// TIA Portal V20 export
// export: Created 2025-12-01T14:57:42.979412Z, ExportSetting None, DisplayName Totally Integrated Automation Portal, DisplayVersion V20 Update 3, DisplayName TIA Portal Openness, DisplayVersion V20 Update 3, DisplayName TIA Portal Version Control Interface, DisplayVersion V20 Update 3, DisplayName STEP 7 Professional, DisplayVersion V20 Update 3, DisplayName STEP 7 Safety, DisplayVersion V20 Update 2, DisplayName WinCC Basic/Comfort/Advanced, DisplayVersion V20 Update 3, DisplayName WinCC Professional, DisplayVersion V20 Update 3, DisplayName WinCC Unified, DisplayVersion V20 Update 3
FUNCTION "FC954_Recoger_Diag_Gateway" : Void   // FC954, LAD
{ S7_Optimized_Access := 'TRUE' }
// stored: AutoNumber false, SetENOAutomatically false
   VAR_TEMP
      i : Int;
      indice : Int;
      datos_gateway : Struct
         Diagnosticar : Bool;   // activar el diagnosticar solo si existe
         Dos_lineas : Bool;
         hwld : HW_IO;
         Dir_ini_diag : Int;
         Dir_ini_Asi5_L1 : Int;
         Dir_ini_ASi5_L2 : Int;
      END_STRUCT;
   END_VAR
BEGIN

REGION Network 1 (SCL)
   // recoger los datos de diagnostico de todos los gateways
   // 
   FOR #indice := 1 TO 8 BY 1 DO
       IF "DB1904_Datos_Config_Gateways".Gateway[#indice].Diagnosticar = true THEN
           #datos_gateway := "DB1904_Datos_Config_Gateways".Gateway[#indice];
           REGION diagnostico_L1
               // diagnostico ASi3- Canal 1
               "DB1903_ASI_DIAG".ASI3_GW_C1[#indice]."Flags Fault Det" := PEEK_WORD(area := 16#1, dbNumber := 0, byteOffset := #datos_gateway.Dir_ini_diag);
               "DB1903_ASI_DIAG".ASI3_GW_C1[#indice].ConfigErrorsW0 := PEEK_WORD(area := 16#1, dbNumber := 0, byteOffset := (#datos_gateway.Dir_ini_diag + 2));
               "DB1903_ASI_DIAG".ASI3_GW_C1[#indice].ConfigErrorsW2 := PEEK_WORD(area := 16#1, dbNumber := 0, byteOffset := (#datos_gateway.Dir_ini_diag + 4));
               "DB1903_ASI_DIAG".ASI3_GW_C1[#indice].ConfigErrorsW4 := PEEK_WORD(area := 16#1, dbNumber := 0, byteOffset := (#datos_gateway.Dir_ini_diag + 6));
               "DB1903_ASI_DIAG".ASI3_GW_C1[#indice].ConfigErrorsW6 := PEEK_WORD(area := 16#1, dbNumber := 0, byteOffset := (#datos_gateway.Dir_ini_diag + 8));
               "DB1903_ASI_DIAG".ASI3_GW_C1[#indice].PeripheryFaultsW0 := PEEK_WORD(area := 16#1, dbNumber := 0, byteOffset := (#datos_gateway.Dir_ini_diag + 10));
               "DB1903_ASI_DIAG".ASI3_GW_C1[#indice].PeripheryFaultsW2 := PEEK_WORD(area := 16#1, dbNumber := 0, byteOffset := (#datos_gateway.Dir_ini_diag + 12));
               "DB1903_ASI_DIAG".ASI3_GW_C1[#indice].PeripheryFaultsW4 := PEEK_WORD(area := 16#1, dbNumber := 0, byteOffset := (#datos_gateway.Dir_ini_diag + 14));
               "DB1903_ASI_DIAG".ASI3_GW_C1[#indice].PeripheryFaultsW6 := PEEK_WORD(area := 16#1, dbNumber := 0, byteOffset := (#datos_gateway.Dir_ini_diag + 16));

               // diagnostico ASi5- Canal 1
               "DB1903_ASI_DIAG".ASI5_GW_C1[#indice].ConfigErrorsW0 := PEEK_WORD(area := 16#1, dbNumber := 0, byteOffset := #datos_gateway.Dir_ini_diag + 18);
               "DB1903_ASI_DIAG".ASI5_GW_C1[#indice].ConfigErrorsW2 := PEEK_WORD(area := 16#1, dbNumber := 0, byteOffset := #datos_gateway.Dir_ini_diag + 20);
               "DB1903_ASI_DIAG".ASI5_GW_C1[#indice].ConfigErrorsW4 := PEEK_WORD(area := 16#1, dbNumber := 0, byteOffset := #datos_gateway.Dir_ini_diag + 22);
               "DB1903_ASI_DIAG".ASI5_GW_C1[#indice].ConfigErrorsW6 := PEEK_WORD(area := 16#1, dbNumber := 0, byteOffset := #datos_gateway.Dir_ini_diag + 24);
               "DB1903_ASI_DIAG".ASI5_GW_C1[#indice].ConfigErrorsW8 := PEEK_WORD(area := 16#1, dbNumber := 0, byteOffset := #datos_gateway.Dir_ini_diag + 26);
               "DB1903_ASI_DIAG".ASI5_GW_C1[#indice].ConfigErrorsW10 := PEEK_WORD(area := 16#1, dbNumber := 0, byteOffset := #datos_gateway.Dir_ini_diag + 28);
               "DB1903_ASI_DIAG".ASI5_GW_C1[#indice].PeripheryFaultsW0 := PEEK_WORD(area := 16#1, dbNumber := 0, byteOffset := #datos_gateway.Dir_ini_diag + 30);
               "DB1903_ASI_DIAG".ASI5_GW_C1[#indice].PeripheryFaultsW2 := PEEK_WORD(area := 16#1, dbNumber := 0, byteOffset := #datos_gateway.Dir_ini_diag + 32);
               "DB1903_ASI_DIAG".ASI5_GW_C1[#indice].PeripheryFaultsW4 := PEEK_WORD(area := 16#1, dbNumber := 0, byteOffset := #datos_gateway.Dir_ini_diag + 34);
               "DB1903_ASI_DIAG".ASI5_GW_C1[#indice].PeripheryFaultsW6 := PEEK_WORD(area := 16#1, dbNumber := 0, byteOffset := #datos_gateway.Dir_ini_diag + 36);
               "DB1903_ASI_DIAG".ASI5_GW_C1[#indice].PeripheryFaultsW8 := PEEK_WORD(area := 16#1, dbNumber := 0, byteOffset := #datos_gateway.Dir_ini_diag + 38);
               "DB1903_ASI_DIAG".ASI5_GW_C1[#indice].PeripheryFaultsW10 := PEEK_WORD(area := 16#1, dbNumber := 0, byteOffset := #datos_gateway.Dir_ini_diag + 40);

               // flags ASi- 5
               "DB1903_ASI_DIAG".ASI5_GW_Flags[#indice].C1_FlagsFault := PEEK_BYTE(area := 16#1, dbNumber := 0, byteOffset := #datos_gateway.Dir_ini_Asi5_L1);

           END_REGION

           REGION diganotico_L2

               IF #datos_gateway.Dos_lineas = true THEN
                   // diagnostico ASi3- Canal 2
                   "DB1903_ASI_DIAG".ASI3_GW_C2[#indice]."Flags Fault Det" := PEEK_WORD(area := 16#1, dbNumber := 0, byteOffset := #datos_gateway.Dir_ini_diag + 42);
                   "DB1903_ASI_DIAG".ASI3_GW_C2[#indice].ConfigErrorsW0 := PEEK_WORD(area := 16#1, dbNumber := 0, byteOffset := #datos_gateway.Dir_ini_diag + 44);
                   "DB1903_ASI_DIAG".ASI3_GW_C2[#indice].ConfigErrorsW2 := PEEK_WORD(area := 16#1, dbNumber := 0, byteOffset := #datos_gateway.Dir_ini_diag + 46);
                   "DB1903_ASI_DIAG".ASI3_GW_C2[#indice].ConfigErrorsW4 := PEEK_WORD(area := 16#1, dbNumber := 0, byteOffset := #datos_gateway.Dir_ini_diag + 48);
                   "DB1903_ASI_DIAG".ASI3_GW_C2[#indice].ConfigErrorsW6 := PEEK_WORD(area := 16#1, dbNumber := 0, byteOffset := #datos_gateway.Dir_ini_diag + 50);
                   "DB1903_ASI_DIAG".ASI3_GW_C2[#indice].PeripheryFaultsW0 := PEEK_WORD(area := 16#1, dbNumber := 0, byteOffset := #datos_gateway.Dir_ini_diag + 52);
                   "DB1903_ASI_DIAG".ASI3_GW_C2[#indice].PeripheryFaultsW2 := PEEK_WORD(area := 16#1, dbNumber := 0, byteOffset := #datos_gateway.Dir_ini_diag + 54);
                   "DB1903_ASI_DIAG".ASI3_GW_C2[#indice].PeripheryFaultsW4 := PEEK_WORD(area := 16#1, dbNumber := 0, byteOffset := #datos_gateway.Dir_ini_diag + 56);
                   "DB1903_ASI_DIAG".ASI3_GW_C2[#indice].PeripheryFaultsW6 := PEEK_WORD(area := 16#1, dbNumber := 0, byteOffset := #datos_gateway.Dir_ini_diag + 58);

                   // diagnostico ASi5- Canal 1
                   "DB1903_ASI_DIAG".ASI5_GW_C2[#indice].ConfigErrorsW0 := PEEK_WORD(area := 16#1, dbNumber := 0, byteOffset := (#datos_gateway.Dir_ini_diag + 60));
                   "DB1903_ASI_DIAG".ASI5_GW_C2[#indice].ConfigErrorsW2 := PEEK_WORD(area := 16#1, dbNumber := 0, byteOffset := #datos_gateway.Dir_ini_diag + 62);
                   "DB1903_ASI_DIAG".ASI5_GW_C2[#indice].ConfigErrorsW4 := PEEK_WORD(area := 16#1, dbNumber := 0, byteOffset := #datos_gateway.Dir_ini_diag + 64);
                   "DB1903_ASI_DIAG".ASI5_GW_C2[#indice].ConfigErrorsW6 := PEEK_WORD(area := 16#1, dbNumber := 0, byteOffset := #datos_gateway.Dir_ini_diag + 66);
                   "DB1903_ASI_DIAG".ASI5_GW_C2[#indice].ConfigErrorsW8 := PEEK_WORD(area := 16#1, dbNumber := 0, byteOffset := #datos_gateway.Dir_ini_diag + 68);
                   "DB1903_ASI_DIAG".ASI5_GW_C2[#indice].ConfigErrorsW10 := PEEK_WORD(area := 16#1, dbNumber := 0, byteOffset := #datos_gateway.Dir_ini_diag + 70);
                   "DB1903_ASI_DIAG".ASI5_GW_C2[#indice].PeripheryFaultsW0 := PEEK_WORD(area := 16#1, dbNumber := 0, byteOffset := #datos_gateway.Dir_ini_diag + 72);
                   "DB1903_ASI_DIAG".ASI5_GW_C2[#indice].PeripheryFaultsW2 := PEEK_WORD(area := 16#1, dbNumber := 0, byteOffset := #datos_gateway.Dir_ini_diag + 74);
                   "DB1903_ASI_DIAG".ASI5_GW_C2[#indice].PeripheryFaultsW4 := PEEK_WORD(area := 16#1, dbNumber := 0, byteOffset := #datos_gateway.Dir_ini_diag + 76);
                   "DB1903_ASI_DIAG".ASI5_GW_C2[#indice].PeripheryFaultsW6 := PEEK_WORD(area := 16#1, dbNumber := 0, byteOffset := #datos_gateway.Dir_ini_diag + 78);
                   "DB1903_ASI_DIAG".ASI5_GW_C2[#indice].PeripheryFaultsW8 := PEEK_WORD(area := 16#1, dbNumber := 0, byteOffset := #datos_gateway.Dir_ini_diag + 80);
                   "DB1903_ASI_DIAG".ASI5_GW_C2[#indice].PeripheryFaultsW10 := PEEK_WORD(area := 16#1, dbNumber := 0, byteOffset := #datos_gateway.Dir_ini_diag + 82);

                   // flags ASi- 5
                   "DB1903_ASI_DIAG".ASI5_GW_Flags[#indice].C2_FlagsFault := PEEK_BYTE(area := 16#1, dbNumber := 0, byteOffset := #datos_gateway.Dir_ini_ASi5_L2);
               END_IF;




           END_REGION

       END_IF;
   END_FOR;
END_REGION
END_FUNCTION
